Staubli VAL3: productionCycle.pgx

program productionCycle()
  local bool l_bPartDone
  local string l_sToolStatus
begin
  // This program is the main cycle. It pick on part from the input
  // conveyor and places it on an empty cavity on the output conveyor.
  //
  // Input parameters
  //  None            :
  //
  // Output parameters
  //  None            :
  //
  //----------------------------------------------------------------
  //
  // In order to improve cycle time, vacuum is always on, even while
  //  placing a part. To place a part, the blow is activated for a
  //  short period of time when the robot arrives to the place position.
  //
  // Main loop

  call getToolStatus(l_sToolStatus)
  if (!bPickDetection and _bPartInTool==true) or (bPickDetection and l_sToolStatus=="PartInTool")
    call place()
  endIf
  //---------------------------------------------------------------------//
  //toRobot1="done"
  do
    //Takes control of the Pick conveyor queue.
    setMutex(_bMutexCnvQueue[0])
    do
      call trackingPick(l_bPartDone)
      delay(0)
    until l_bPartDone
    // Release control of the Pick conveyor queue.
    _bMutexCnvQueue[0]=false

    //
    call place()
    //
    delay(0)
  until _bEndCycle
  _bEndCycle=true
  //
end
